{region '#Template'}
	{attribute 'Version' := '5.0.0.0'}
	{attribute 'Tags' := '"LCID": "1031", "Text": "Universal, Sensor, BI"'}
	{attribute 'Tags' := '"LCID": "1033", "Text": "Universal, Sensor, BI"'}
	{attribute 'Using' := '"Type": "Template", "URI": "EC_ID"'}
	{attribute 'Using' := '"Type": "Template", "URI": "BA2_Param"'}
	{attribute 'Description' := '"LCID": "1031", "Text": "BI mit IO"'}
	{attribute 'Description' := '"LCID": "1033", "Text": "BI with IO"'}
{endregion}		 
FUNCTION_BLOCK FB_BA_SensorBinary_Raw EXTENDS FB_BA_View
VAR_INPUT
END_VAR
VAR_INPUT CONSTANT
	Input					: FB_BA_BI_Raw;		
END_VAR
VAR_OUTPUT
	bPresentValue			: BOOL;	
END_VAR
VAR
END_VAR

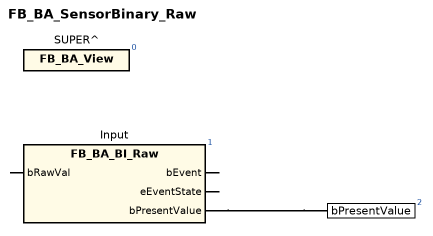
SUPER^(); // FB_BA_View
Input(); // FB_BA_BI_Raw
bPresentValue := Input.bPresentValue;

METHOD FB_init : BOOL
VAR_INPUT
	bInitRetains : BOOL; // if TRUE, the retain variables are initialized (warm start / cold start)
	bInCopyCode : BOOL;  // if TRUE, the instance afterwards gets moved into the copy code (online change)
END_VAR
Input.iParent						:= THIS^;
Input.iLabel						:= LblFun_Fault;
Input.ePolarity						:= E_BA_Polarity.eReverse;
Input.sActiveText 					:= txtEvent_Triggered;
Input.sInactiveText 				:= txtEvent_Normal;
Input.nEventClassID					:= EC_ID.NC30;
Input.stTimeDelay.nToNormal			:= BA2_Param.nDefTimeDelay_ToNormal;
Input.stTimeDelay.nToAbnormal		:= BA2_Param.nDefTimeDelay_ToAbnormal;
Input.bAlarmValue					:= TRUE;
Input.aEventTransitionText[1]		:= txtEvent_Triggered;
Input.aEventTransitionText[2]		:= txtEvent_Error;
Input.aEventTransitionText[3]		:= txtEvent_Normal;
Input.bEventDetectionEnable			:= TRUE;
Input.eEnPlantLock					:= E_BA_LockPriority.eNoLock;
END_METHOD

END_FUNCTION_BLOCK

(* stored: Version 1.1.0.1, ProductVersion 3.1.4024.12
   POU FB_BA_SensorBinary_Raw: Id {707cb882-1d24-4a73-879a-43bdde016831}, SpecialFunc None
   Method FB_init: Id {2dbb9e34-6250-448e-8ddc-49479a7d4711} *)
